Omron CX-Programmer project NewProject (CX-Programmer 9.73)

# PLC NewPLC1: CP1E E30

## Global symbols (name address type ; comment)
100.05 BOOL  ; G3 down
10.02 BOOL  ; set G3 down
0.05 BOOL  ; sensor F
T009 BOOL  ; delay G3 down
100.04 BOOL  ; G3 up
T007 BOOL  ; delay G3 up
0.04 BOOL  ; sensor E
100.03 BOOL  ; G2 down
10.01 BOOL  ; set G2 down
T006 BOOL  ; delay G2 down
100.02 BOOL  ; G2 up
T004 BOOL  ; delay G2 up
100.01 BOOL  ; G1 down
10.00 BOOL  ; set G1 down
T002 BOOL  ; delay G1 down
100.00 BOOL  ; G1 up
T000 BOOL  ; delay G1 up
0.03 BOOL  ; sensor D
0.02 BOOL  ; sensor C
0.01 BOOL  ; sensor B
0.00 BOOL  ; sensor A
100.06 BOOL  ; V1 penuh
100.07 BOOL  ; V2 penuh
D1 CHANNEL  ; data V1
D2 CHANNEL  ; data V2
T001 BOOL  ; delay set G1 down
T005 BOOL  ; delay set G2 down
T008 BOOL  ; delay set G3 down
W0.01 BOOL  ; M.V1
W0.02 BOOL  ; M.V2

## Program NewProgram1 (cyclic task 0)

### Section Section1

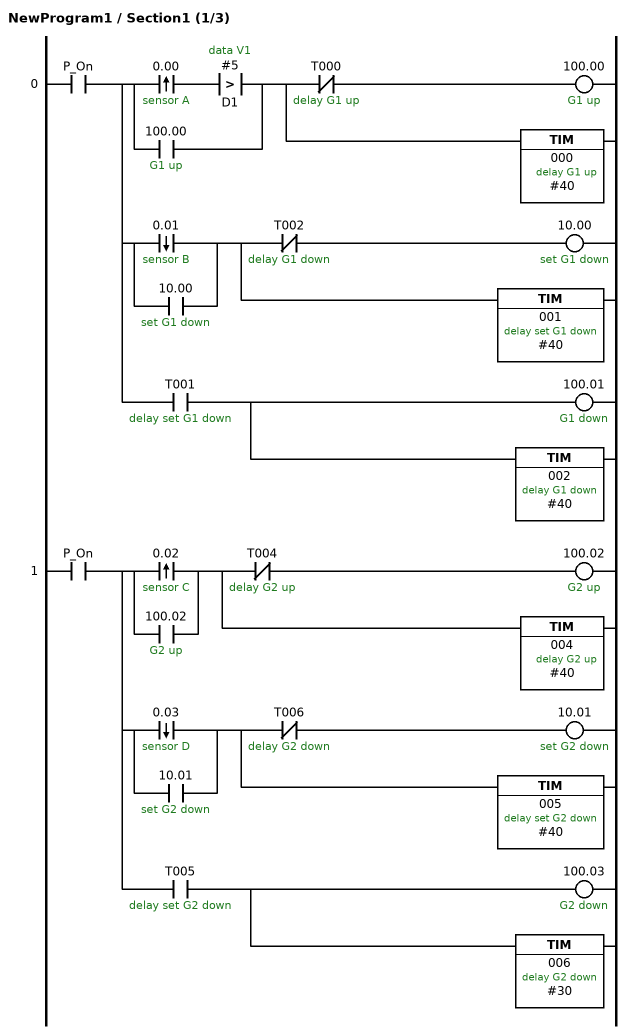
; rung 0
LD P_On
OUT TR0
@LD 0.00  ; sensor A
AND>(320) #5 D1  ; data V1
OR 100.00  ; G1 up
ANDLD
OUT TR1
ANDNOT T000  ; delay G1 up
OUT 100.00  ; G1 up
LD TR1
TIM 000 #40  ; delay G1 up
LD TR0
%LD 0.01  ; sensor B
OR 10.00  ; set G1 down
ANDLD
OUT TR1
ANDNOT T002  ; delay G1 down
OUT 10.00  ; set G1 down
LD TR1
TIM 001 #40  ; delay set G1 down
LD TR0
AND T001  ; delay set G1 down
OUT 100.01  ; G1 down
TIM 002 #40  ; delay G1 down
; rung 1
LD P_On
OUT TR0
@LD 0.02  ; sensor C
OR 100.02  ; G2 up
ANDLD
OUT TR1
ANDNOT T004  ; delay G2 up
OUT 100.02  ; G2 up
LD TR1
TIM 004 #40  ; delay G2 up
LD TR0
%LD 0.03  ; sensor D
OR 10.01  ; set G2 down
ANDLD
OUT TR1
ANDNOT T006  ; delay G2 down
OUT 10.01  ; set G2 down
LD TR1
TIM 005 #40  ; delay set G2 down
LD TR0
AND T005  ; delay set G2 down
OUT 100.03  ; G2 down
TIM 006 #30  ; delay G2 down

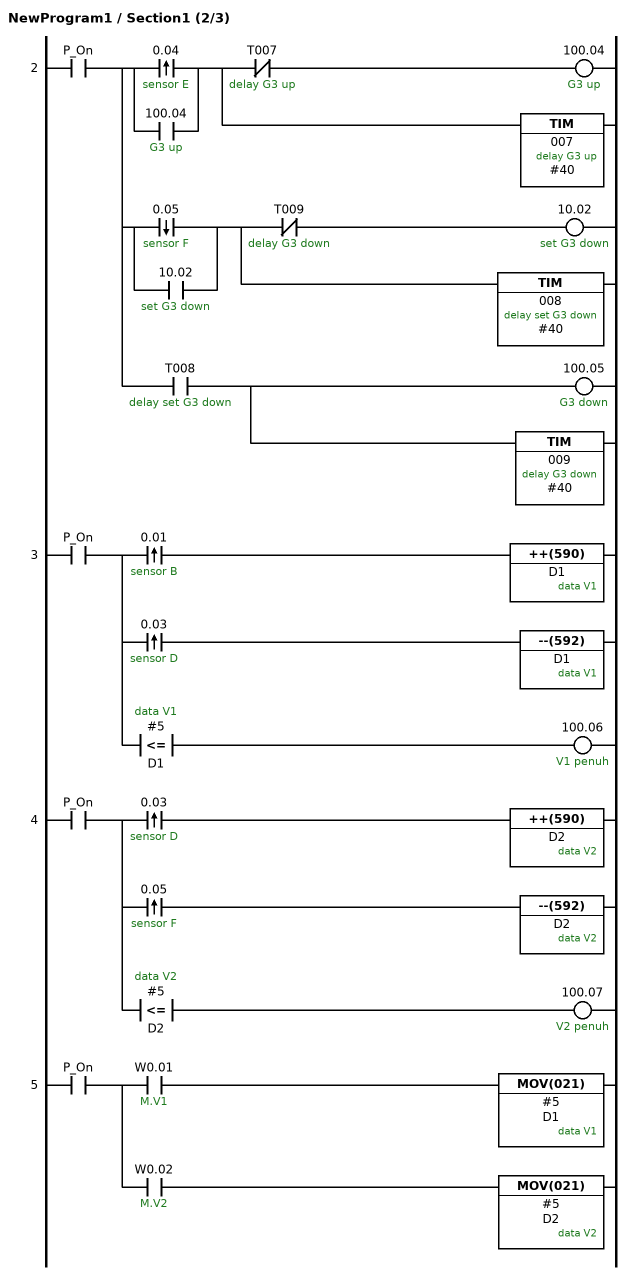
; rung 2
LD P_On
OUT TR0
@LD 0.04  ; sensor E
OR 100.04  ; G3 up
ANDLD
OUT TR1
ANDNOT T007  ; delay G3 up
OUT 100.04  ; G3 up
LD TR1
TIM 007 #40  ; delay G3 up
LD TR0
%LD 0.05  ; sensor F
OR 10.02  ; set G3 down
ANDLD
OUT TR1
ANDNOT T009  ; delay G3 down
OUT 10.02  ; set G3 down
LD TR1
TIM 008 #40  ; delay set G3 down
LD TR0
AND T008  ; delay set G3 down
OUT 100.05  ; G3 down
TIM 009 #40  ; delay G3 down
; rung 3
LD P_On
OUT TR0
@AND 0.01  ; sensor B
++(590) D1  ; data V1
LD TR0
@AND 0.03  ; sensor D
--(592) D1  ; data V1
LD TR0
AND<=(315) #5 D1  ; data V1
OUT 100.06  ; V1 penuh
; rung 4
LD P_On
OUT TR0
@AND 0.03  ; sensor D
++(590) D2  ; data V2
LD TR0
@AND 0.05  ; sensor F
--(592) D2  ; data V2
LD TR0
AND<=(315) #5 D2  ; data V2
OUT 100.07  ; V2 penuh
; rung 5
LD P_On
OUT TR0
AND W0.01  ; M.V1
MOV(021) #5 D1  ; data V1
LD TR0
AND W0.02  ; M.V2
MOV(021) #5 D2  ; data V2

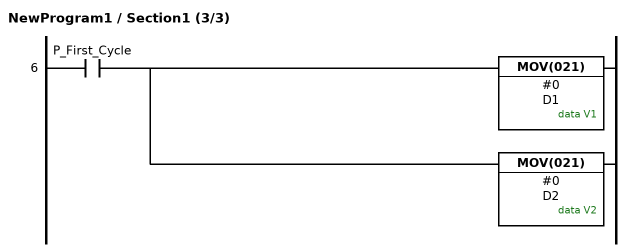
; rung 6
LD P_First_Cycle
MOV(021) #0 D1  ; data V1
MOV(021) #0 D2  ; data V2

### Section END
; rung 0
END(001)